// This function has been automatically generated from the project information.
VAR_GLOBAL CONSTANT
	{attribute 'const_non_replaced'}
	stLibVersion_Base_Hts : ST_LibVersion := (iMajor := 0, iMinor := 0, iBuild := 1, iRevision := 0, sVersion := '0.0.1.0');
END_VAR

(* stored: Version 1.1.0.1, ProductVersion 3.1.0.36
   GVL Global_Version: Id {b736f4d7-b848-4c63-89cf-5a896f3db631} *)
